FUNCTION_BLOCK FB_SearchString
VAR_INPUT
	Person    : Pers_data; //DUT STRUCT
	SearchTxt : STRING(25);
END_VAR
VAR_OUTPUT
	Match     : BOOL;
END_VAR
VAR
	AllText   : STRING(120);
	AllTextLower  : STRING(120);
	SearchLower   : STRING(25);
END_VAR

(* alles samenvoegen *)
AllText := CONCAT(
				CONCAT(Person.Name, Person.Firstname),
				Person.Address
			);

(* naar lowercase omzetten *)
AllTextLower := F_ToLCase(AllText);
SearchLower  := F_ToLCase(SearchTxt);

(* vergelijken *)
IF FIND(AllTextLower, SearchLower) > 0 THEN
	Match := TRUE;
ELSE
	Match := FALSE;
END_IF

END_FUNCTION_BLOCK

(* stored: Version 1.1.0.1, ProductVersion 3.1.4024.15
   POU FB_SearchString: Id {0d1ccf8d-19c5-4c5b-82eb-72f5881f243d}, SpecialFunc None *)
